FUNCTION_BLOCK PUBLIC FB_AmericanPizzaMargherita EXTENDS FB_PizzaAmericanStyle
VAR_INPUT
END_VAR
VAR_OUTPUT
END_VAR
VAR
	bCheese		: BOOL := TRUE;
	bTomato		: BOOL := TRUE;
END_VAR

PROPERTY PUBLIC bHasCheese : BOOL
GET
bHasCheese := this^.bCheese;
END_GET
SET
this^.bCheese := bHasCheese;
END_SET
END_PROPERTY

PROPERTY PUBLIC bHasTomato : BOOL
GET
bHasTomato := this^.bTomato;
END_GET
SET
this^.bTomato := bHasTomato;
END_SET
END_PROPERTY

METHOD PUBLIC GetPrice : LREAL
VAR_INPUT
END_VAR
GetPrice := SUPER^.GetPrice();
IF (THIS^.bCheese) THEN
	GetPrice := GetPrice + 1.1;
END_IF
IF (THIS^.bTomato) THEN
	GetPrice := GetPrice + 0.9;
END_IF
END_METHOD

END_FUNCTION_BLOCK

(* stored: Version 1.1.0.1, ProductVersion 3.1.4022.12
   POU FB_AmericanPizzaMargherita: Id {25b1758a-210d-44bc-8d7c-06295dec0eb4}, SpecialFunc None
   Property bHasCheese: Id {a8bd2b21-a7de-4a3a-b58d-a9f95e94f964}
   Get Get: Id {46307bed-5059-4905-bcf8-cb87239ceb0e}
   Set Set: Id {6a3a6266-8d89-4739-b4cd-d1c0986fa6b2}
   Property bHasTomato: Id {d108d26d-f265-4e2e-8eac-27ac1a6105ed}
   Get Get: Id {e6ebf1bc-c809-44f7-aa62-307e17b96fb9}
   Set Set: Id {a77f01bc-5fa7-45c9-80a1-6a74ff3eb04c}
   Method GetPrice: Id {06a1782b-9249-40a7-9973-4e645f31797f} *)
